// TwinCAT 3 PLC project PipelineTests
// ProgramVersion: 3.1.4026.22
// libraries:
//   Tc2_Standard, * (Beckhoff Automation GmbH)
//   Tc2_System, * (Beckhoff Automation GmbH)
//   TcUnit, * (www.tcunit.org)
//   B4Pipeline_Plc,newest,Tc3 Project
// project tree:
//   / PlcTask.TcTTO
//   POUs/ FB_PipelineConsumer.TcPOU, MAIN.TcPOU
// real-time tasks:
//   TASK PlcTask: cycle T#10ms, priority 20, ADS port 350

CONFIGURATION PipelineTests
    RESOURCE PLC ON TwinCAT3
        TASK PlcTask(INTERVAL := T#10ms, PRIORITY := 20);
        PROGRAM MAIN WITH PlcTask : MAIN;
    END_RESOURCE
END_CONFIGURATION

// ---- POUs/MAIN.TcPOU
PROGRAM MAIN
VAR
END_VAR

END_PROGRAM

// ---- POUs/FB_PipelineConsumer.TcPOU
FUNCTION_BLOCK FB_PipelineConsumer
VAR
    stage : B4Pipeline_Plc.FB_PipelineStage;
    bStageError : BOOL;
END_VAR

stage(value := -1);
bStageError := stage.bError;

END_FUNCTION_BLOCK
